{attribute 'qualified_only'}
{attribute 'strict'}
{attribute 'to_string'}
TYPE MACHINE_STATE :
(
	BOOTING := 0,
	ABORTING,
	ABORTED,
	CLEARING,
	COMPLETING, 
	COMPLETE, 
	EXECUTING,
	HOLDING,
	HELD,
	IDLE,
	RESETTING,
	STARTING,
	STOPPING,
	STOPPED,
	SUSPENDING,
	SUSPENDED,
	UNHOLDING,
	UNSUSPENDING,
	END	
);
END_TYPE

(* stored: Version 1.1.0.1
   EnumerationTextList MACHINE_STATE: Id {d757ed78-d646-43a3-80b6-9c2b7ba77cfc} *)
